{attribute addProperty BoxType "EP8309-0022-0021"}
{attribute addProperty Id "Digital_Output_X4_Pin4AT %Q*BOOL811Digital_Output_X4_Pin2AT %Q*BOOL812Digital_Output_X5_Pin4AT %Q*BOOL813Digital_Output_X5_Pin2AT %Q*BOOL814Digital_Output_X6_Pin4AT %Q*BOOL815Digital_Output_X6_Pin2AT %Q*BOOL816Digital_Output_X7_Pin4AT %Q*BOOL817Digital_Output_X7_Pin2AT %Q*BOOL818"}
{attribute addProperty CRC "3071836906"}
{attribute addProperty SizeInBites "64"}
{attribute addProperty SizeInBytes "8"}
TYPE DIG_Outputs_B71882EA :
STRUCT
	{attribute addProperty Name "Digital_Output_X4_Pin4"}
	Digital_Output_X4_Pin4 AT %Q* : BOOL;
	{attribute addProperty Name "Digital_Output_X4_Pin2"}
	Digital_Output_X4_Pin2 AT %Q* : BOOL;
	{attribute addProperty Name "Digital_Output_X5_Pin4"}
	Digital_Output_X5_Pin4 AT %Q* : BOOL;
	{attribute addProperty Name "Digital_Output_X5_Pin2"}
	Digital_Output_X5_Pin2 AT %Q* : BOOL;
	{attribute addProperty Name "Digital_Output_X6_Pin4"}
	Digital_Output_X6_Pin4 AT %Q* : BOOL;
	{attribute addProperty Name "Digital_Output_X6_Pin2"}
	Digital_Output_X6_Pin2 AT %Q* : BOOL;
	{attribute addProperty Name "Digital_Output_X7_Pin4"}
	Digital_Output_X7_Pin4 AT %Q* : BOOL;
	{attribute addProperty Name "Digital_Output_X7_Pin2"}
	Digital_Output_X7_Pin2 AT %Q* : BOOL;
END_STRUCT
END_TYPE

(* stored: Version 1.2.0.0, ProductVersion 3.1.4024.9
   DUT DIG_Outputs_B71882EA: Id {60ef60f0-342e-4d99-9d84-575711a8f3a9} *)
